FUNCTION_BLOCK FB_TimestampRegistryTest
VAR_INPUT
END_VAR
VAR_OUTPUT
END_VAR
VAR
END_VAR

END_FUNCTION_BLOCK

(* stored: Version 1.1.0.1, ProductVersion 3.1.4024.12
   POU FB_TimestampRegistryTest: Id {dc36b022-c4cc-4e93-ada4-75afce70000f}, SpecialFunc None *)
